{attribute 'linkalways'} 
{attribute 'no_explicit_call' := 'This FB is a CLASS and must be accessed using methods or properties'}
{attribute 'enable_dynamic_creation'}
FUNCTION_BLOCK _ETcVnOcrModelType EXTENDS EnumDatatypeBase
VAR
	localData : ETcVnOcrModelType;
	activeData : REFERENCE TO ETcVnOcrModelType;
	enumBaseDatatype : _ULINT(localData);
END_VAR

METHOD PRIVATE AddLocalEnumeration
VAR_INPUT
	Enumeration : T_MAXSTRING;
	Value : ETcVnOcrModelType;
END_VAR
AddEnumeration(Enumeration, Value);
END_METHOD

PROPERTY PUBLIC Address : PVOID
GET
Address := ADR(activeData);
END_GET
END_PROPERTY

METHOD PUBLIC ClearReference
VAR_INPUT
END_VAR
activeData REF= localData;
SetBaseDatatypeReference();
END_METHOD

METHOD PUBLIC Clone : I_Datatype
VAR
    pClone : POINTER TO _ETcVnOcrModelType;
END_VAR
pClone := __NEW(_ETcVnOcrModelType(InitialValue := Value));
Clone := pClone^;
END_METHOD

METHOD FB_init : BOOL
VAR_INPUT
	bInitRetains : BOOL; // if TRUE, the retain variables are initialized (warm start / cold start)
	bInCopyCode : BOOL;  // if TRUE, the instance afterwards gets moved into the copy code (online change)
	InitialValue : ETcVnOcrModelType;
END_VAR
localData := InitialValue;
AddBaseDatatype(enumBaseDatatype);
ClearReference();

AddLocalEnumeration('TCVN_OMT_NUMBERS', ETcVnOcrModelType.TCVN_OMT_NUMBERS);
AddLocalEnumeration('TCVN_OMT_NUMBERS_SC', ETcVnOcrModelType.TCVN_OMT_NUMBERS_SC);
AddLocalEnumeration('TCVN_OMT_UCLETTERS', ETcVnOcrModelType.TCVN_OMT_UCLETTERS);
AddLocalEnumeration('TCVN_OMT_NUMBERS_SC_UCLETTERS', ETcVnOcrModelType.TCVN_OMT_NUMBERS_SC_UCLETTERS);
AddLocalEnumeration('TCVN_OMT_CNN_NUMBERS_SC_LETTERS', ETcVnOcrModelType.TCVN_OMT_CNN_NUMBERS_SC_LETTERS);
END_METHOD

PROPERTY PUBLIC Identifier : T_MAXSTRING
GET
Identifier := 'ETcVnOcrModelType';
END_GET
END_PROPERTY

METHOD IsEnumeratorValueEqual : BOOL
VAR_INPUT
	Enumerator : I_KeyValueForwardEnumerator;
END_VAR
VAR
	storedValue : ETcVnOcrModelType;
END_VAR
IF NOT Enumerator.TryGet(storedValue) THEN
	RETURN;
END_IF

IsEnumeratorValueEqual := storedValue = activeData;
END_METHOD

METHOD PUBLIC MakeReferenceTo
VAR_INPUT
	ReferenceTarget : REFERENCE TO ETcVnOcrModelType;
END_VAR
activeData REF= ReferenceTarget;
SetBaseDatatypeReference();
END_METHOD

METHOD PROTECTED SetBaseDatatypeReference
VAR_INPUT
END_VAR
enumBaseDatatype.MakeReferenceTo(activeData);
END_METHOD

PROPERTY PUBLIC Size : UDINT
GET
Size := SIZEOF(activeData);
END_GET
END_PROPERTY

METHOD TryMakeReferenceTo : BOOL
VAR_INPUT
	Target : I_Datatype;
END_VAR
VAR
	pTargetData : POINTER TO ETcVnOcrModelType;
END_VAR
IF NOT IsEquivalentTo(Target) THEN
	RETURN;
END_IF

pTargetData := Target.Address;
activeData REF= pTargetData^;
SetBaseDatatypeReference();
TryMakeReferenceTo := TRUE;
END_METHOD

PROPERTY PUBLIC Value : ETcVnOcrModelType
GET
Value := activeData;
END_GET
SET
activeData := Value;
END_SET
END_PROPERTY

END_FUNCTION_BLOCK

(* stored: Version 1.1.0.1, ProductVersion 3.1.4024.13
   POU _ETcVnOcrModelType: Id {31c59095-d60a-056c-02e4-ee62e1839971}, SpecialFunc None
   Folder Core: Id {9775bda9-047f-0f3c-27af-9272b56c24c7}
   Folder Protected: Id {1d322fdd-1e01-011a-26d3-5a6aeea3bc2e}
   Folder Customize: Id {f6af8425-3d67-01ba-3562-43b9f23b244b}
   Folder Constructor: Id {e4da3c75-c518-0532-1729-e64a23f45243}
   Folder Private: Id {64fcf79b-acda-0dda-2716-04b49b9ea99c}
   Folder Protected: Id {13b9b73e-4a05-0b02-29e3-01c633ceb6b3}
   Method AddLocalEnumeration: Id {74acef2b-2f7f-0a15-0611-be6dfd8f816b}
   Property Address: Id {7df267e5-58e2-0164-177c-a0ea18caf922}
   Get Get: Id {72737d9f-047e-067f-3a23-c216ca943b61}
   Method ClearReference: Id {e326594e-6a56-0a2c-0037-1577a53da7c0}
   Method Clone: Id {ac1087f7-450c-0481-0766-402cc32ff53d}
   Method FB_init: Id {7a8c9ca5-0c53-0f58-27cf-9f69d1fcaa1b}
   Property Identifier: Id {24d9adde-8027-028a-19ac-aabc22ca699f}
   Get Get: Id {1e580ce9-1e23-0f28-2b8f-6e64212dbeba}
   Method IsEnumeratorValueEqual: Id {b3b63983-6a27-0db8-097e-1eed67c1699e}
   Method MakeReferenceTo: Id {fab4a4d1-f638-0089-2d49-b3b832e9a8f7}
   Method SetBaseDatatypeReference: Id {41a63a24-210a-01a3-1395-55917d3edeb8}
   Property Size: Id {781eef86-2082-0214-328c-1ca1f4657922}
   Get Get: Id {d644c06f-1bac-0c1d-264e-bc39877f20c5}
   Method TryMakeReferenceTo: Id {4de3a9b2-e89b-0312-217f-ffceda9b7972}
   Property Value: Id {6694afbd-725e-0095-3a3d-c54ebf28e10f}
   Get Get: Id {d84e773b-6a84-0f26-3e5d-a93d65344229}
   Set Set: Id {a6b79dbf-0ccb-0f91-22a3-7130e0358876} *)
